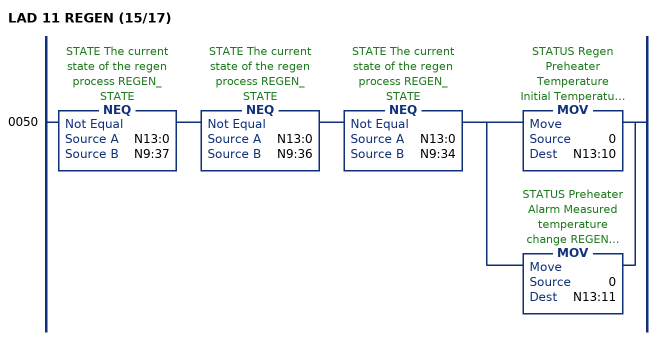
% Rung: 50 %
SOR NEQ N13:0 N9:37 NEQ N13:0 N9:36 NEQ N13:0 N9:34 BST MOV 0 N13:10 NXB MOV 0 N13:11 BND EOR
%   N13:0  REGEN_STATE  "STATE The current state of the regen process" %
%   N9:37  REGEN_ALARM  "STATE Regen Alarm" %
%   N9:36  REGEN_COOL  "STATE Regen Cool" %
%   N9:34  REGEN_RUN  "STATE Regen Running" %
%   N13:10  REGEN_HRS_LEFT  "STATUS Regen Preheater Temperature Initial Temperature" %
%   N13:11  REGEN_MIN_LEFT  "STATUS Preheater Alarm Measured temperature change" %

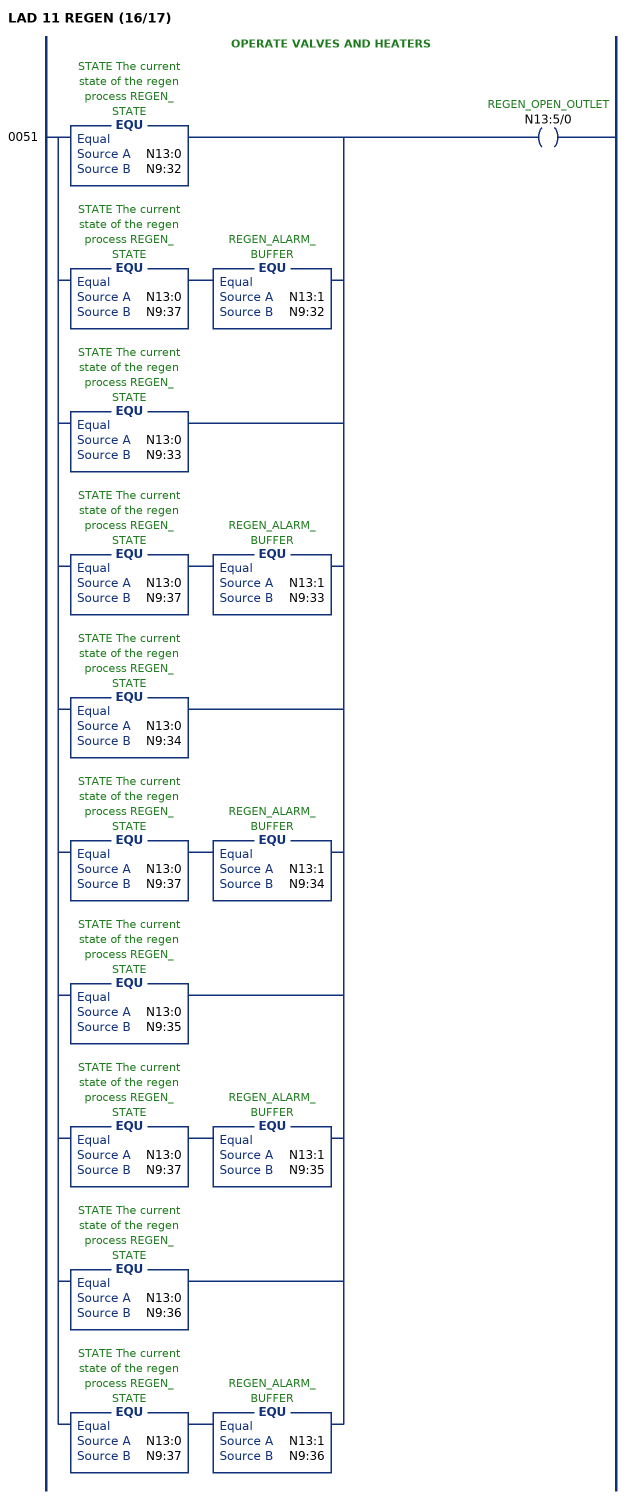
% Rung: 51 %
% TITLE: OPERATE VALVES AND HEATERS %
SOR BST EQU N13:0 N9:32 NXB EQU N13:0 N9:37 EQU N13:1 N9:32 NXB EQU N13:0 N9:33 NXB EQU N13:0 N9:37 EQU N13:1 N9:33 NXB EQU N13:0 N9:34 NXB EQU N13:0 N9:37 EQU N13:1 N9:34 NXB EQU N13:0 N9:35 NXB EQU N13:0 N9:37 EQU N13:1 N9:35 NXB EQU N13:0 N9:36 NXB EQU N13:0 N9:37 EQU N13:1 N9:36 BND OTE N13:5/0 EOR
%   N13:0  REGEN_STATE  "STATE The current state of the regen process" %
%   N9:32  REGEN_VENT  "STATE Regen Vent" %
%   N9:37  REGEN_ALARM  "STATE Regen Alarm" %
%   N13:1  REGEN_ALARM_BUFFER %
%   N9:33  REGEN_HEAT_BED  "STATE Regen Heat wall" %
%   N9:34  REGEN_RUN  "STATE Regen Running" %
%   N9:35  REGEN_COOL_WALL  "STATE Regen Cool wall" %
%   N9:36  REGEN_COOL  "STATE Regen Cool" %
%   N13:5/0  REGEN_OPEN_OUTLET %

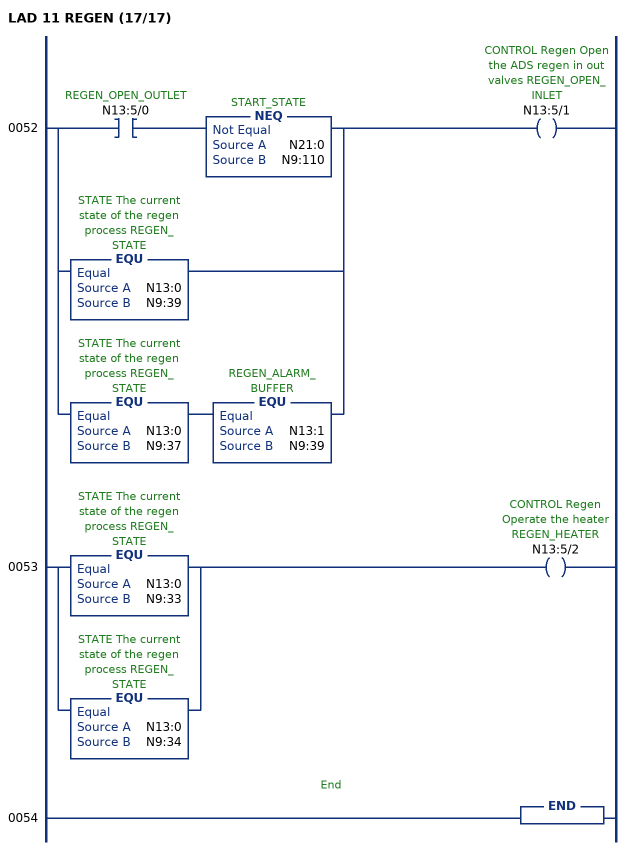
% Rung: 52 %
SOR BST XIC N13:5/0 NEQ N21:0 N9:110 NXB EQU N13:0 N9:39 NXB EQU N13:0 N9:37 EQU N13:1 N9:39 BND OTE N13:5/1 EOR
%   N13:5/0  REGEN_OPEN_OUTLET %
%   N21:0  START_STATE %
%   N9:110  START_REG_VENT %
%   N13:0  REGEN_STATE  "STATE The current state of the regen process" %
%   N9:39  REGEN_BACKFILL %
%   N9:37  REGEN_ALARM  "STATE Regen Alarm" %
%   N13:1  REGEN_ALARM_BUFFER %
%   N13:5/1  REGEN_OPEN_INLET  "CONTROL Regen Open the ADS regen in out valves" %
% Rung: 53 %
SOR BST EQU N13:0 N9:33 NXB EQU N13:0 N9:34 BND OTE N13:5/2 EOR
%   N13:0  REGEN_STATE  "STATE The current state of the regen process" %
%   N9:33  REGEN_HEAT_BED  "STATE Regen Heat wall" %
%   N9:34  REGEN_RUN  "STATE Regen Running" %
%   N13:5/2  REGEN_HEATER  "CONTROL Regen Operate the heater" %
% Rung: 54 %
% End %
SOR END EOR

LADDER 12 "REGEN_FLT"    % regen alarms and warnings %
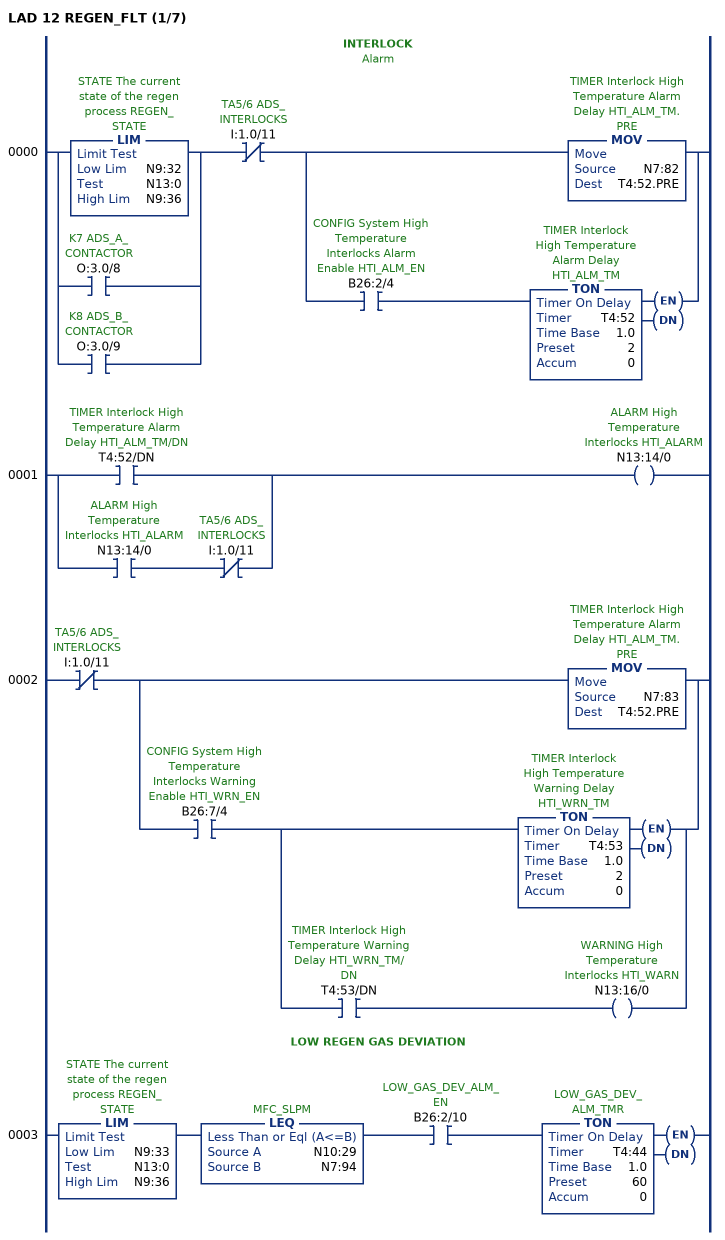
% Rung: 0 %
% TITLE: INTERLOCK %
% Alarm %
SOR BST LIM N9:32 N13:0 N9:36 NXB XIC O:3.0/8 NXB XIC O:3.0/9 BND XIO I:1.0/11 BST MOV N7:82 T4:52.PRE NXB XIC B26:2/4 TON T4:52 1.0 2 0 BND EOR
%   N9:32  REGEN_VENT  "STATE Regen Vent" %
%   N13:0  REGEN_STATE  "STATE The current state of the regen process" %
%   N9:36  REGEN_COOL  "STATE Regen Cool" %
%   O:3.0/8  ADS_A_CONTACTOR  "K7" %
%   O:3.0/9  ADS_B_CONTACTOR  "K8" %
%   I:1.0/11  ADS_INTERLOCKS  "TA5/6" %
%   N7:82  HTI_ALM_DY  "CONFIG Interlocks High Temp Alarm Delay" %
%   T4:52  HTI_ALM_TM  "TIMER Interlock High Temperature Alarm Delay" %
%   B26:2/4  HTI_ALM_EN  "CONFIG System High Temperature Interlocks Alarm Enable" %
% Rung: 1 %
SOR BST XIC T4:52/DN NXB XIC N13:14/0 XIO I:1.0/11 BND OTE N13:14/0 EOR
%   T4:52  HTI_ALM_TM  "TIMER Interlock High Temperature Alarm Delay" %
%   N13:14/0  HTI_ALARM  "ALARM High Temperature Interlocks" %
%   I:1.0/11  ADS_INTERLOCKS  "TA5/6" %
% Rung: 2 %
SOR XIO I:1.0/11 BST MOV N7:83 T4:52.PRE NXB XIC B26:7/4 BST TON T4:53 1.0 2 0 NXB XIC T4:53/DN OTE N13:16/0 BND BND EOR
%   I:1.0/11  ADS_INTERLOCKS  "TA5/6" %
%   N7:83  HTI_WRN_DY  "CONFIG Interlocks High Temp Warning Delay" %
%   T4:52  HTI_ALM_TM  "TIMER Interlock High Temperature Alarm Delay" %
%   B26:7/4  HTI_WRN_EN  "CONFIG System High Temperature Interlocks Warning Enable" %
%   T4:53  HTI_WRN_TM  "TIMER Interlock High Temperature Warning Delay" %
%   N13:16/0  HTI_WARN  "WARNING High Temperature Interlocks" %
% Rung: 3 %
% TITLE: LOW REGEN GAS DEVIATION %
SOR LIM N9:33 N13:0 N9:36 LEQ N10:29 N7:94 XIC B26:2/10 TON T4:44 1.0 60 0 EOR
%   N9:33  REGEN_HEAT_BED  "STATE Regen Heat wall" %
%   N13:0  REGEN_STATE  "STATE The current state of the regen process" %
%   N9:36  REGEN_COOL  "STATE Regen Cool" %
%   N10:29  MFC_SLPM %
%   N7:94  LOW_GAS_DEV_ALM_SP %
%   B26:2/10  LOW_GAS_DEV_ALM_EN %
%   T4:44  LOW_GAS_DEV_ALM_TMR %

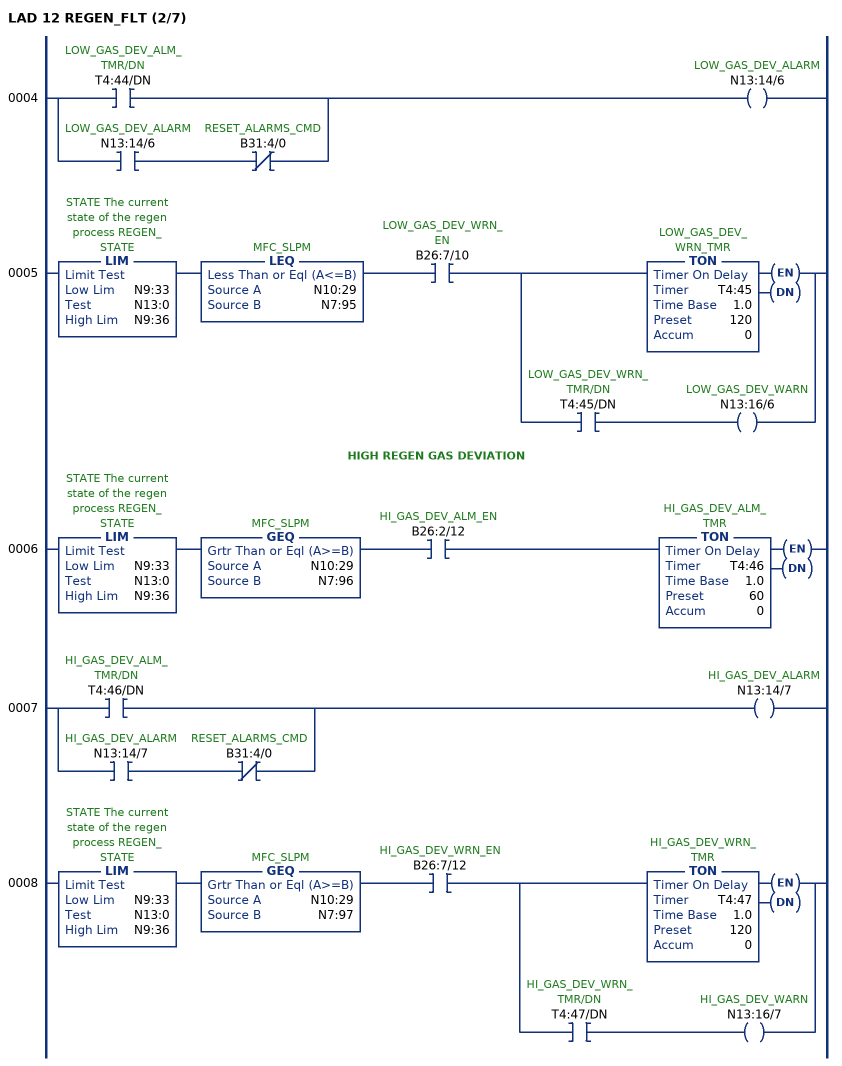
% Rung: 4 %
SOR BST XIC T4:44/DN NXB XIC N13:14/6 XIO B31:4/0 BND OTE N13:14/6 EOR
%   T4:44  LOW_GAS_DEV_ALM_TMR %
%   N13:14/6  LOW_GAS_DEV_ALARM %
%   B31:4/0  RESET_ALARMS_CMD %
% Rung: 5 %
SOR LIM N9:33 N13:0 N9:36 LEQ N10:29 N7:95 XIC B26:7/10 BST TON T4:45 1.0 120 0 NXB XIC T4:45/DN OTE N13:16/6 BND EOR
%   N9:33  REGEN_HEAT_BED  "STATE Regen Heat wall" %
%   N13:0  REGEN_STATE  "STATE The current state of the regen process" %
%   N9:36  REGEN_COOL  "STATE Regen Cool" %
%   N10:29  MFC_SLPM %
%   N7:95  LOW_GAS_DEV_WRN_SP %
%   B26:7/10  LOW_GAS_DEV_WRN_EN %
%   T4:45  LOW_GAS_DEV_WRN_TMR %
%   N13:16/6  LOW_GAS_DEV_WARN %
% Rung: 6 %
% TITLE: HIGH REGEN GAS DEVIATION %
SOR LIM N9:33 N13:0 N9:36 GEQ N10:29 N7:96 XIC B26:2/12 TON T4:46 1.0 60 0 EOR
%   N9:33  REGEN_HEAT_BED  "STATE Regen Heat wall" %
%   N13:0  REGEN_STATE  "STATE The current state of the regen process" %
%   N9:36  REGEN_COOL  "STATE Regen Cool" %
%   N10:29  MFC_SLPM %
%   N7:96  HI_GAS_DEV_ALM_SP %
%   B26:2/12  HI_GAS_DEV_ALM_EN %
%   T4:46  HI_GAS_DEV_ALM_TMR %
% Rung: 7 %
SOR BST XIC T4:46/DN NXB XIC N13:14/7 XIO B31:4/0 BND OTE N13:14/7 EOR
%   T4:46  HI_GAS_DEV_ALM_TMR %
%   N13:14/7  HI_GAS_DEV_ALARM %
%   B31:4/0  RESET_ALARMS_CMD %
% Rung: 8 %
SOR LIM N9:33 N13:0 N9:36 GEQ N10:29 N7:97 XIC B26:7/12 BST TON T4:47 1.0 120 0 NXB XIC T4:47/DN OTE N13:16/7 BND EOR
%   N9:33  REGEN_HEAT_BED  "STATE Regen Heat wall" %
%   N13:0  REGEN_STATE  "STATE The current state of the regen process" %
%   N9:36  REGEN_COOL  "STATE Regen Cool" %
%   N10:29  MFC_SLPM %
%   N7:97  HI_GAS_DEV_WRN_SP %
%   B26:7/12  HI_GAS_DEV_WRN_EN %
%   T4:47  HI_GAS_DEV_WRN_TMR %
%   N13:16/7  HI_GAS_DEV_WARN %

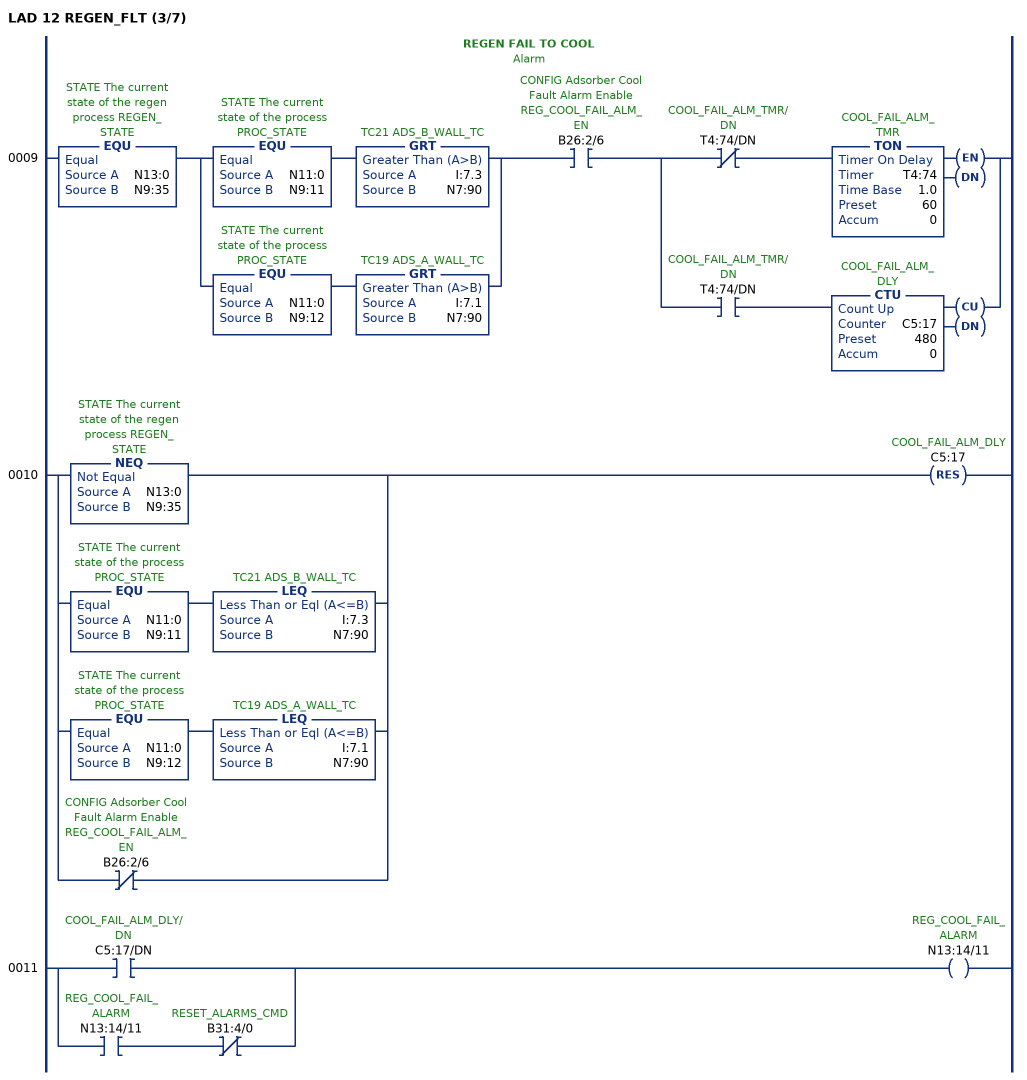
% Rung: 9 %
% TITLE: REGEN FAIL TO COOL %
% Alarm %
SOR EQU N13:0 N9:35 BST EQU N11:0 N9:11 GRT I:7.3 N7:90 NXB EQU N11:0 N9:12 GRT I:7.1 N7:90 BND XIC B26:2/6 BST XIO T4:74/DN TON T4:74 1.0 60 0 NXB XIC T4:74/DN CTU C5:17 480 0 BND EOR
%   N13:0  REGEN_STATE  "STATE The current state of the regen process" %
%   N9:35  REGEN_COOL_WALL  "STATE Regen Cool wall" %
%   N11:0  PROC_STATE  "STATE The current state of the process" %
%   N9:11  PROC_PFY_A_REG_B  "STATE Process Purify A" %
%   I:7.3  ADS_B_WALL_TC  "TC21" %
%   N7:90  REG_COOL_FAIL_ALM_SP %
%   N9:12  PROC_PFY_B_REG_A  "STATE Process Purify B" %
%   I:7.1  ADS_A_WALL_TC  "TC19" %
%   B26:2/6  REG_COOL_FAIL_ALM_EN  "CONFIG Adsorber Cool Fault Alarm Enable" %
%   T4:74  COOL_FAIL_ALM_TMR %
%   C5:17  COOL_FAIL_ALM_DLY %
% Rung: 10 %
SOR BST NEQ N13:0 N9:35 NXB EQU N11:0 N9:11 LEQ I:7.3 N7:90 NXB EQU N11:0 N9:12 LEQ I:7.1 N7:90 NXB XIO B26:2/6 BND RES C5:17 EOR
%   N13:0  REGEN_STATE  "STATE The current state of the regen process" %
%   N9:35  REGEN_COOL_WALL  "STATE Regen Cool wall" %
%   N11:0  PROC_STATE  "STATE The current state of the process" %
%   N9:11  PROC_PFY_A_REG_B  "STATE Process Purify A" %
%   I:7.3  ADS_B_WALL_TC  "TC21" %
%   N7:90  REG_COOL_FAIL_ALM_SP %
%   N9:12  PROC_PFY_B_REG_A  "STATE Process Purify B" %
%   I:7.1  ADS_A_WALL_TC  "TC19" %
%   B26:2/6  REG_COOL_FAIL_ALM_EN  "CONFIG Adsorber Cool Fault Alarm Enable" %
%   C5:17  COOL_FAIL_ALM_DLY %
% Rung: 11 %
SOR BST XIC C5:17/DN NXB XIC N13:14/11 XIO B31:4/0 BND OTE N13:14/11 EOR
%   C5:17  COOL_FAIL_ALM_DLY %
%   N13:14/11  REG_COOL_FAIL_ALARM %
%   B31:4/0  RESET_ALARMS_CMD %

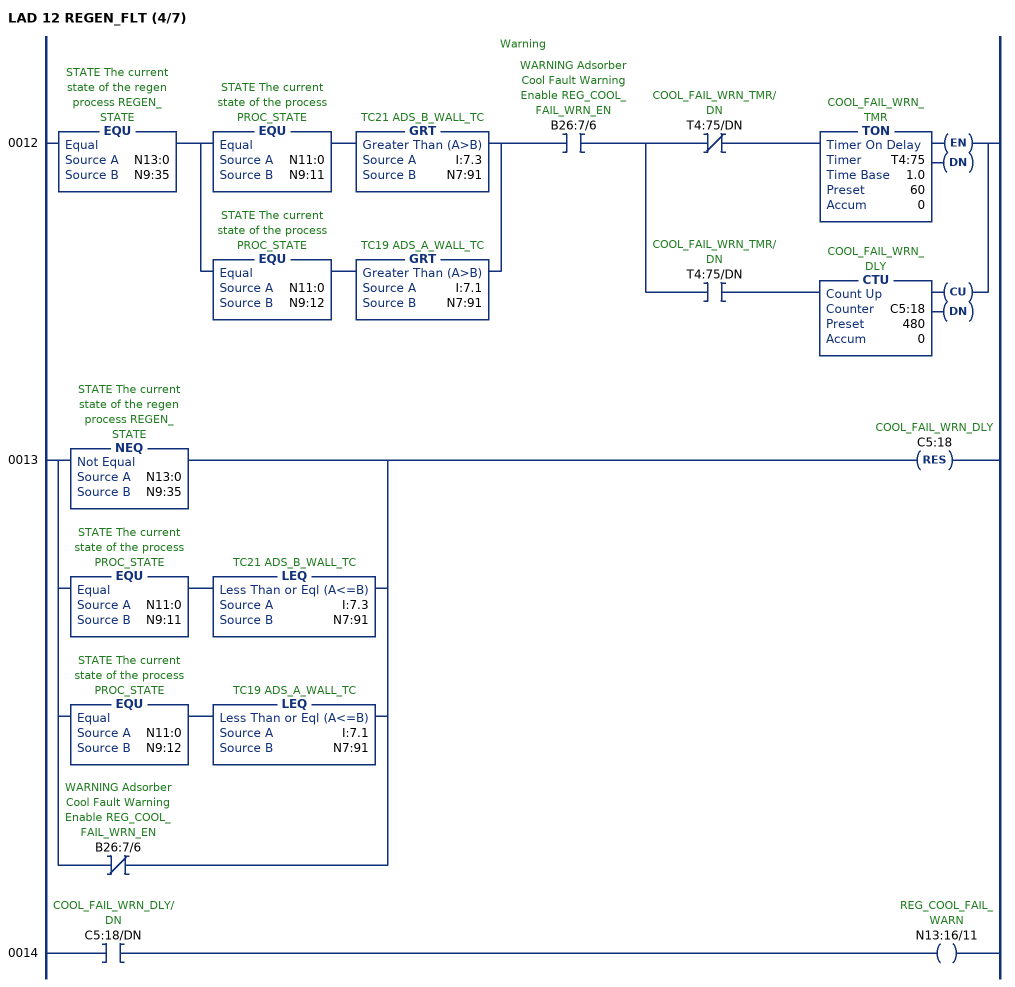
% Rung: 12 %
% Warning %
SOR EQU N13:0 N9:35 BST EQU N11:0 N9:11 GRT I:7.3 N7:91 NXB EQU N11:0 N9:12 GRT I:7.1 N7:91 BND XIC B26:7/6 BST XIO T4:75/DN TON T4:75 1.0 60 0 NXB XIC T4:75/DN CTU C5:18 480 0 BND EOR
%   N13:0  REGEN_STATE  "STATE The current state of the regen process" %
%   N9:35  REGEN_COOL_WALL  "STATE Regen Cool wall" %
%   N11:0  PROC_STATE  "STATE The current state of the process" %
%   N9:11  PROC_PFY_A_REG_B  "STATE Process Purify A" %
%   I:7.3  ADS_B_WALL_TC  "TC21" %
%   N7:91  REG_COOL_FAIL_WRN_SP %
%   N9:12  PROC_PFY_B_REG_A  "STATE Process Purify B" %
%   I:7.1  ADS_A_WALL_TC  "TC19" %
%   B26:7/6  REG_COOL_FAIL_WRN_EN  "WARNING Adsorber Cool Fault Warning Enable" %
%   T4:75  COOL_FAIL_WRN_TMR %
%   C5:18  COOL_FAIL_WRN_DLY %
% Rung: 13 %
SOR BST NEQ N13:0 N9:35 NXB EQU N11:0 N9:11 LEQ I:7.3 N7:91 NXB EQU N11:0 N9:12 LEQ I:7.1 N7:91 NXB XIO B26:7/6 BND RES C5:18 EOR
%   N13:0  REGEN_STATE  "STATE The current state of the regen process" %
%   N9:35  REGEN_COOL_WALL  "STATE Regen Cool wall" %
%   N11:0  PROC_STATE  "STATE The current state of the process" %
%   N9:11  PROC_PFY_A_REG_B  "STATE Process Purify A" %
%   I:7.3  ADS_B_WALL_TC  "TC21" %
%   N7:91  REG_COOL_FAIL_WRN_SP %
%   N9:12  PROC_PFY_B_REG_A  "STATE Process Purify B" %
%   I:7.1  ADS_A_WALL_TC  "TC19" %
%   B26:7/6  REG_COOL_FAIL_WRN_EN  "WARNING Adsorber Cool Fault Warning Enable" %
%   C5:18  COOL_FAIL_WRN_DLY %
% Rung: 14 %
SOR XIC C5:18/DN OTE N13:16/11 EOR
%   C5:18  COOL_FAIL_WRN_DLY %
%   N13:16/11  REG_COOL_FAIL_WARN %

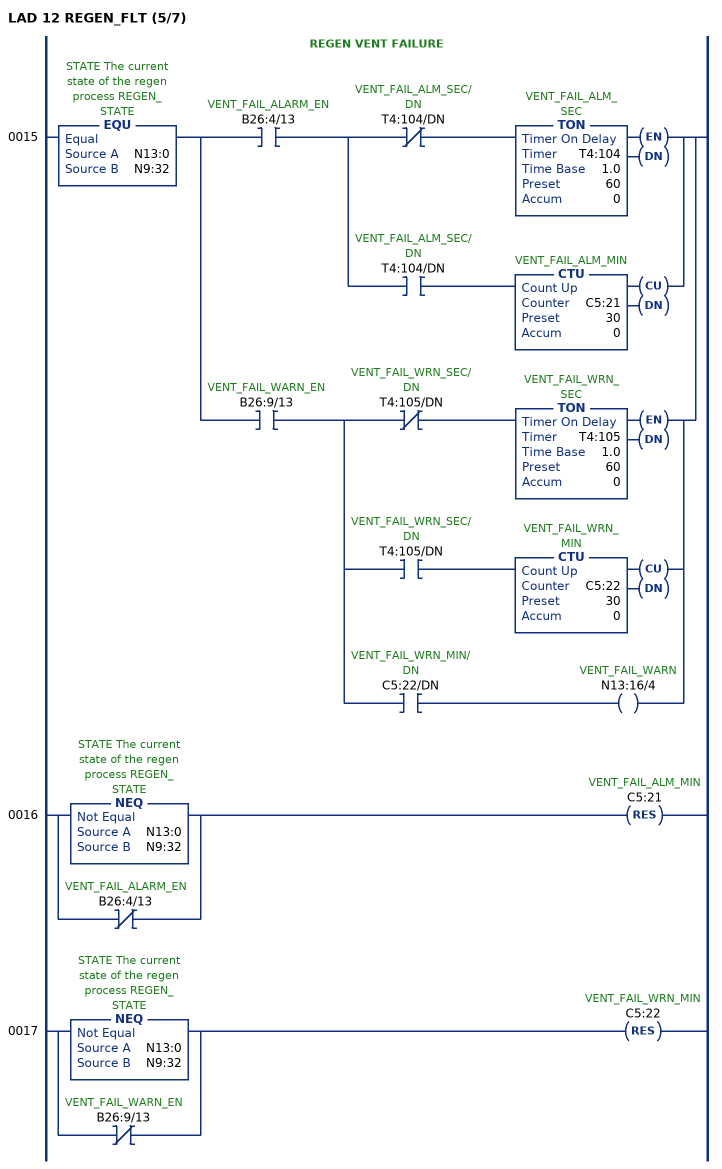
% Rung: 15 %
% TITLE: REGEN VENT FAILURE %
SOR EQU N13:0 N9:32 BST XIC B26:4/13 BST XIO T4:104/DN TON T4:104 1.0 60 0 NXB XIC T4:104/DN CTU C5:21 30 0 BND NXB XIC B26:9/13 BST XIO T4:105/DN TON T4:105 1.0 60 0 NXB XIC T4:105/DN CTU C5:22 30 0 NXB XIC C5:22/DN OTE N13:16/4 BND BND EOR
%   N13:0  REGEN_STATE  "STATE The current state of the regen process" %
%   N9:32  REGEN_VENT  "STATE Regen Vent" %
%   B26:4/13  VENT_FAIL_ALARM_EN %
%   T4:104  VENT_FAIL_ALM_SEC %
%   C5:21  VENT_FAIL_ALM_MIN %
%   B26:9/13  VENT_FAIL_WARN_EN %
%   T4:105  VENT_FAIL_WRN_SEC %
%   C5:22  VENT_FAIL_WRN_MIN %
%   N13:16/4  VENT_FAIL_WARN %
% Rung: 16 %
SOR BST NEQ N13:0 N9:32 NXB XIO B26:4/13 BND RES C5:21 EOR
%   N13:0  REGEN_STATE  "STATE The current state of the regen process" %
%   N9:32  REGEN_VENT  "STATE Regen Vent" %
%   B26:4/13  VENT_FAIL_ALARM_EN %
%   C5:21  VENT_FAIL_ALM_MIN %
% Rung: 17 %
SOR BST NEQ N13:0 N9:32 NXB XIO B26:9/13 BND RES C5:22 EOR
%   N13:0  REGEN_STATE  "STATE The current state of the regen process" %
%   N9:32  REGEN_VENT  "STATE Regen Vent" %
%   B26:9/13  VENT_FAIL_WARN_EN %
%   C5:22  VENT_FAIL_WRN_MIN %

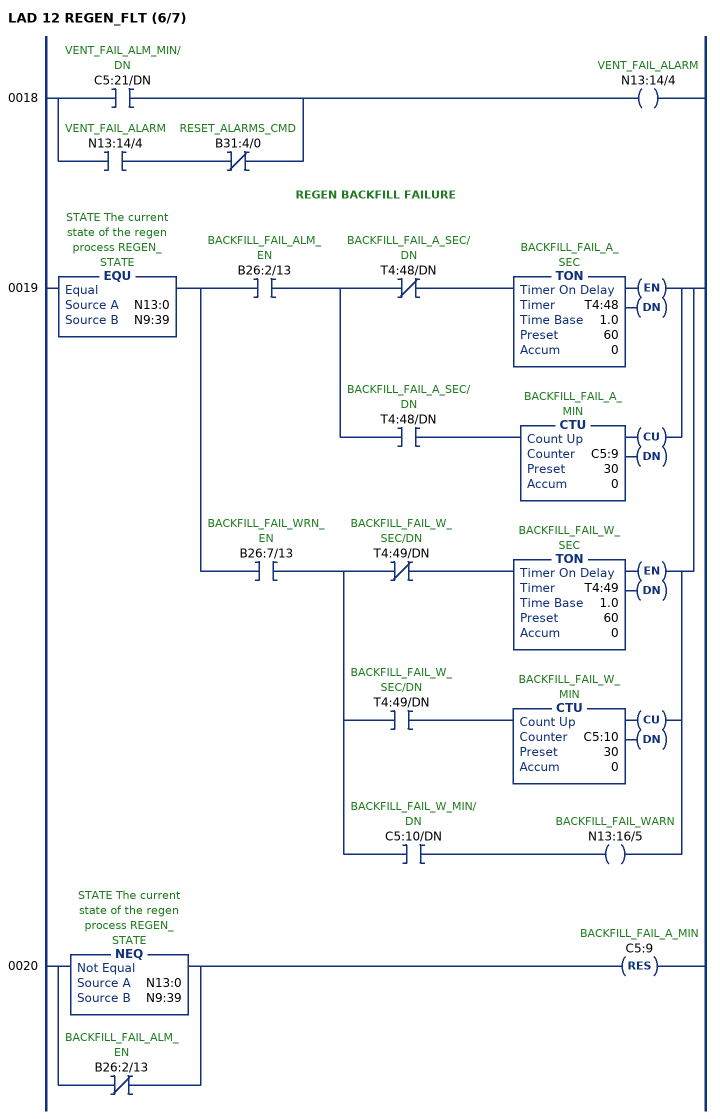
% Rung: 18 %
SOR BST XIC C5:21/DN NXB XIC N13:14/4 XIO B31:4/0 BND OTE N13:14/4 EOR
%   C5:21  VENT_FAIL_ALM_MIN %
%   N13:14/4  VENT_FAIL_ALARM %
%   B31:4/0  RESET_ALARMS_CMD %
% Rung: 19 %
% TITLE: REGEN BACKFILL FAILURE %
SOR EQU N13:0 N9:39 BST XIC B26:2/13 BST XIO T4:48/DN TON T4:48 1.0 60 0 NXB XIC T4:48/DN CTU C5:9 30 0 BND NXB XIC B26:7/13 BST XIO T4:49/DN TON T4:49 1.0 60 0 NXB XIC T4:49/DN CTU C5:10 30 0 NXB XIC C5:10/DN OTE N13:16/5 BND BND EOR
%   N13:0  REGEN_STATE  "STATE The current state of the regen process" %
%   N9:39  REGEN_BACKFILL %
%   B26:2/13  BACKFILL_FAIL_ALM_EN %
%   T4:48  BACKFILL_FAIL_A_SEC %
%   C5:9  BACKFILL_FAIL_A_MIN %
%   B26:7/13  BACKFILL_FAIL_WRN_EN %
%   T4:49  BACKFILL_FAIL_W_SEC %
%   C5:10  BACKFILL_FAIL_W_MIN %
%   N13:16/5  BACKFILL_FAIL_WARN %
% Rung: 20 %
SOR BST NEQ N13:0 N9:39 NXB XIO B26:2/13 BND RES C5:9 EOR
%   N13:0  REGEN_STATE  "STATE The current state of the regen process" %
%   N9:39  REGEN_BACKFILL %
%   B26:2/13  BACKFILL_FAIL_ALM_EN %
%   C5:9  BACKFILL_FAIL_A_MIN %

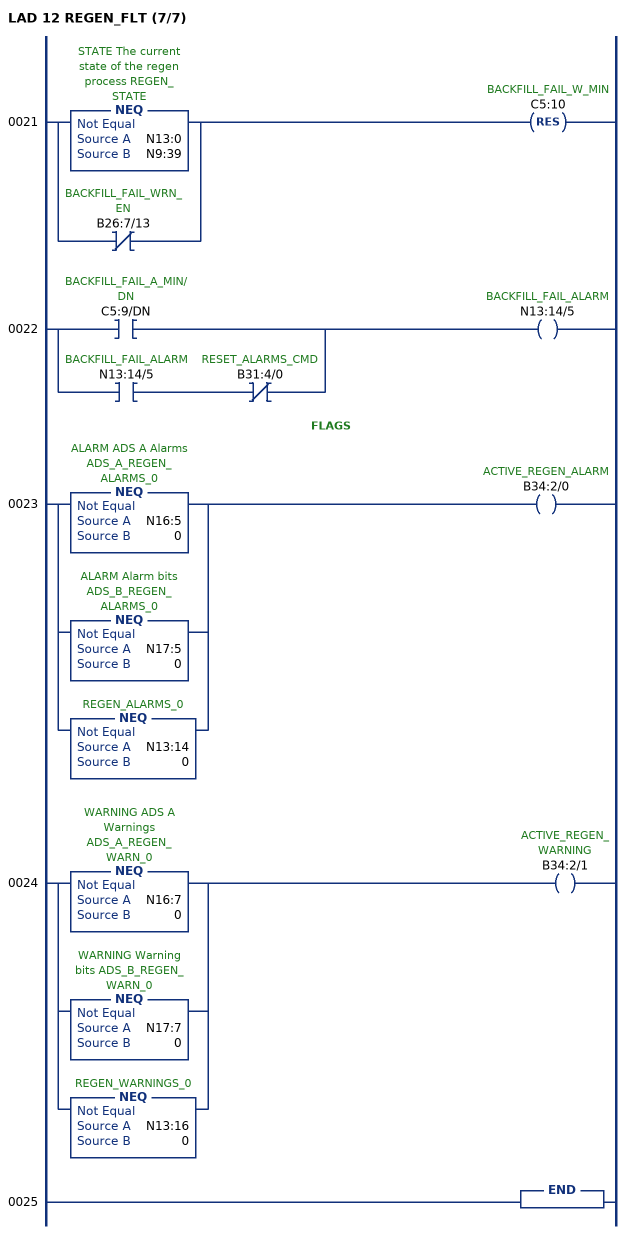
% Rung: 21 %
SOR BST NEQ N13:0 N9:39 NXB XIO B26:7/13 BND RES C5:10 EOR
%   N13:0  REGEN_STATE  "STATE The current state of the regen process" %
%   N9:39  REGEN_BACKFILL %
%   B26:7/13  BACKFILL_FAIL_WRN_EN %
%   C5:10  BACKFILL_FAIL_W_MIN %
% Rung: 22 %
SOR BST XIC C5:9/DN NXB XIC N13:14/5 XIO B31:4/0 BND OTE N13:14/5 EOR
%   C5:9  BACKFILL_FAIL_A_MIN %
%   N13:14/5  BACKFILL_FAIL_ALARM %
%   B31:4/0  RESET_ALARMS_CMD %
% Rung: 23 %
% TITLE: FLAGS %
SOR BST NEQ N16:5 0 NXB NEQ N17:5 0 NXB NEQ N13:14 0 BND OTE B34:2/0 EOR
%   N16:5  ADS_A_REGEN_ALARMS_0  "ALARM ADS A Alarms" %
%   N17:5  ADS_B_REGEN_ALARMS_0  "ALARM Alarm bits" %
%   N13:14  REGEN_ALARMS_0 %
%   B34:2/0  ACTIVE_REGEN_ALARM %
% Rung: 24 %
SOR BST NEQ N16:7 0 NXB NEQ N17:7 0 NXB NEQ N13:16 0 BND OTE B34:2/1 EOR
%   N16:7  ADS_A_REGEN_WARN_0  "WARNING ADS A Warnings" %
%   N17:7  ADS_B_REGEN_WARN_0  "WARNING Warning bits" %
%   N13:16  REGEN_WARNINGS_0 %
%   B34:2/1  ACTIVE_REGEN_WARNING %
% Rung: 25 %
SOR END EOR

LADDER 13 "PURGE"
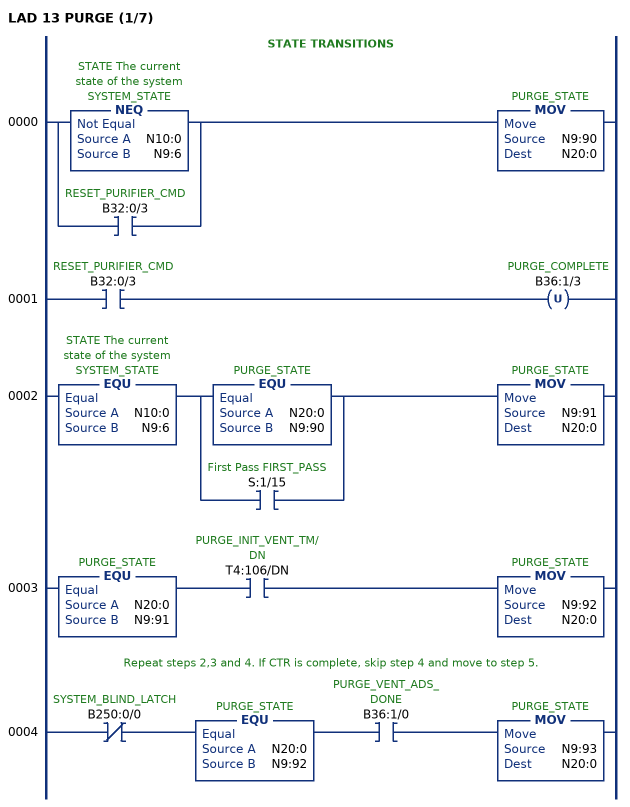
% Rung: 0 %
% TITLE: STATE TRANSITIONS %
SOR BST NEQ N10:0 N9:6 NXB XIC B32:0/3 BND MOV N9:90 N20:0 EOR
%   N10:0  SYSTEM_STATE  "STATE The current state of the system" %
%   N9:6  SYSTEM_PURGE %
%   B32:0/3  RESET_PURIFIER_CMD %
%   N9:90  PURGE_IDLE %
%   N20:0  PURGE_STATE %
% Rung: 1 %
SOR XIC B32:0/3 OTU B36:1/3 EOR
%   B32:0/3  RESET_PURIFIER_CMD %
%   B36:1/3  PURGE_COMPLETE %
% Rung: 2 %
SOR EQU N10:0 N9:6 BST EQU N20:0 N9:90 NXB XIC S:1/15 BND MOV N9:91 N20:0 EOR
%   N10:0  SYSTEM_STATE  "STATE The current state of the system" %
%   N9:6  SYSTEM_PURGE %
%   N20:0  PURGE_STATE %
%   N9:90  PURGE_IDLE %
%   S:1/15  FIRST_PASS  "First Pass" %
%   N9:91  PURGE_INIT_VENT %
% Rung: 3 %
SOR EQU N20:0 N9:91 XIC T4:106/DN MOV N9:92 N20:0 EOR
%   N20:0  PURGE_STATE %
%   N9:91  PURGE_INIT_VENT %
%   T4:106  PURGE_INIT_VENT_TM %
%   N9:92  PURGE_VENT_ADSORBER %
% Rung: 4 %
% Repeat steps 2,3 and 4. If CTR is complete, skip step 4 and move to step 5. %
SOR XIO B250:0/0 EQU N20:0 N9:92 XIC B36:1/0 MOV N9:93 N20:0 EOR
%   B250:0/0  SYSTEM_BLIND_LATCH %
%   N20:0  PURGE_STATE %
%   N9:92  PURGE_VENT_ADSORBER %
%   B36:1/0  PURGE_VENT_ADS_DONE %
%   N9:93  PURGE_VENT_GETTER %

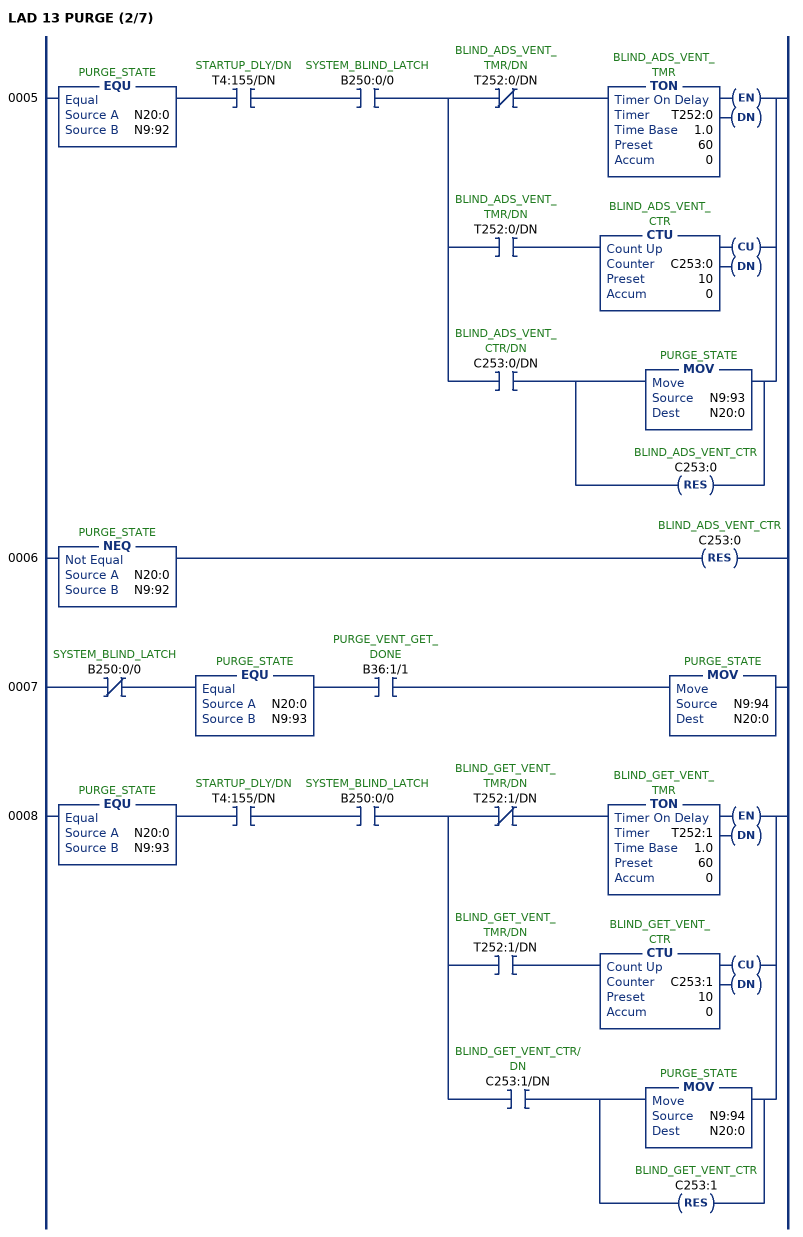
% Rung: 5 %
SOR EQU N20:0 N9:92 XIC T4:155/DN XIC B250:0/0 BST XIO T252:0/DN TON T252:0 1.0 60 0 NXB XIC T252:0/DN CTU C253:0 10 0 NXB XIC C253:0/DN BST MOV N9:93 N20:0 NXB RES C253:0 BND BND EOR
%   N20:0  PURGE_STATE %
%   N9:92  PURGE_VENT_ADSORBER %
%   T4:155  STARTUP_DLY %
%   B250:0/0  SYSTEM_BLIND_LATCH %
%   T252:0  BLIND_ADS_VENT_TMR %
%   C253:0  BLIND_ADS_VENT_CTR %
%   N9:93  PURGE_VENT_GETTER %
% Rung: 6 %
SOR NEQ N20:0 N9:92 RES C253:0 EOR
%   N20:0  PURGE_STATE %
%   N9:92  PURGE_VENT_ADSORBER %
%   C253:0  BLIND_ADS_VENT_CTR %
% Rung: 7 %
SOR XIO B250:0/0 EQU N20:0 N9:93 XIC B36:1/1 MOV N9:94 N20:0 EOR
%   B250:0/0  SYSTEM_BLIND_LATCH %
%   N20:0  PURGE_STATE %
%   N9:93  PURGE_VENT_GETTER %
%   B36:1/1  PURGE_VENT_GET_DONE %
%   N9:94  PURGE_BACKFILL %
% Rung: 8 %
SOR EQU N20:0 N9:93 XIC T4:155/DN XIC B250:0/0 BST XIO T252:1/DN TON T252:1 1.0 60 0 NXB XIC T252:1/DN CTU C253:1 10 0 NXB XIC C253:1/DN BST MOV N9:94 N20:0 NXB RES C253:1 BND BND EOR
%   N20:0  PURGE_STATE %
%   N9:93  PURGE_VENT_GETTER %
%   T4:155  STARTUP_DLY %
%   B250:0/0  SYSTEM_BLIND_LATCH %
%   T252:1  BLIND_GET_VENT_TMR %
%   C253:1  BLIND_GET_VENT_CTR %
%   N9:94  PURGE_BACKFILL %

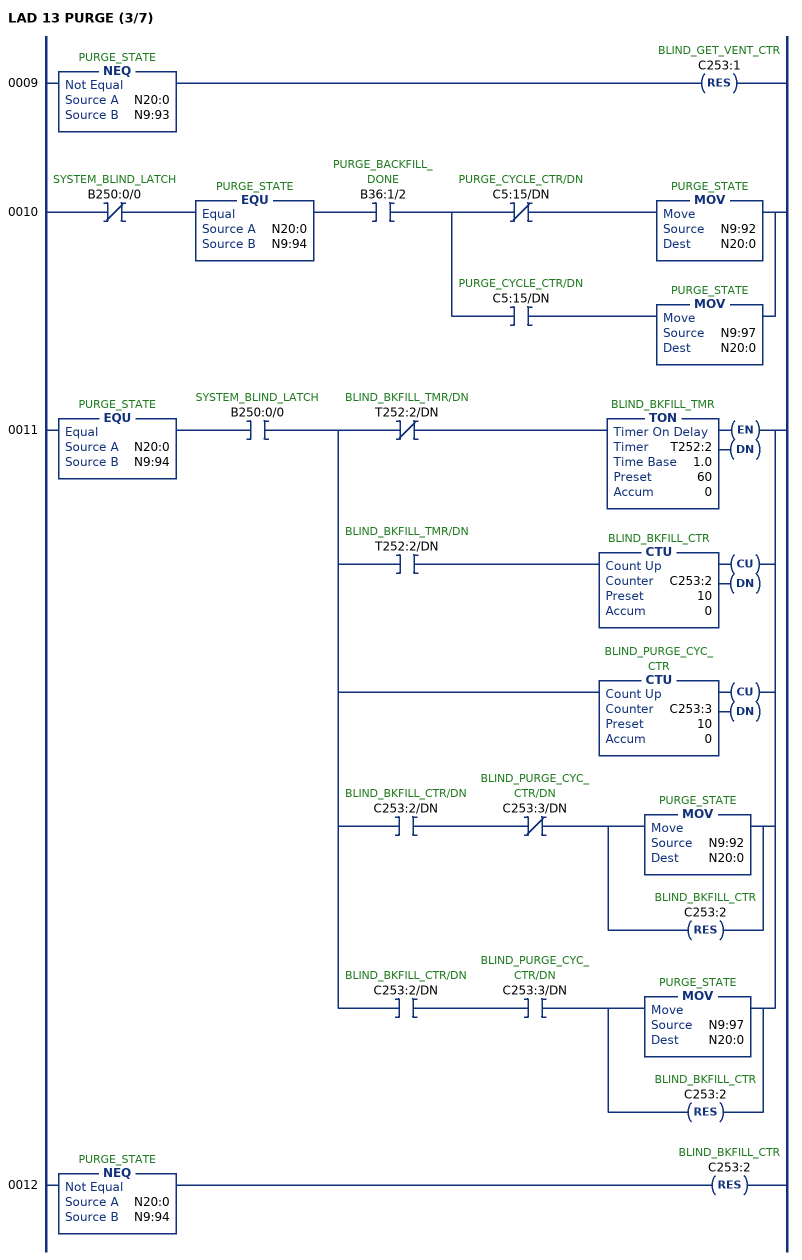
% Rung: 9 %
SOR NEQ N20:0 N9:93 RES C253:1 EOR
%   N20:0  PURGE_STATE %
%   N9:93  PURGE_VENT_GETTER %
%   C253:1  BLIND_GET_VENT_CTR %
% Rung: 10 %
SOR XIO B250:0/0 EQU N20:0 N9:94 XIC B36:1/2 BST XIO C5:15/DN MOV N9:92 N20:0 NXB XIC C5:15/DN MOV N9:97 N20:0 BND EOR
%   B250:0/0  SYSTEM_BLIND_LATCH %
%   N20:0  PURGE_STATE %
%   N9:94  PURGE_BACKFILL %
%   B36:1/2  PURGE_BACKFILL_DONE %
%   C5:15  PURGE_CYCLE_CTR %
%   N9:92  PURGE_VENT_ADSORBER %
%   N9:97  PURGE_VENT_ADS_2 %
% Rung: 11 %
SOR EQU N20:0 N9:94 XIC B250:0/0 BST XIO T252:2/DN TON T252:2 1.0 60 0 NXB XIC T252:2/DN CTU C253:2 10 0 NXB CTU C253:3 10 0 NXB XIC C253:2/DN XIO C253:3/DN BST MOV N9:92 N20:0 NXB RES C253:2 BND NXB XIC C253:2/DN XIC C253:3/DN BST MOV N9:97 N20:0 NXB RES C253:2 BND BND EOR
%   N20:0  PURGE_STATE %
%   N9:94  PURGE_BACKFILL %
%   B250:0/0  SYSTEM_BLIND_LATCH %
%   T252:2  BLIND_BKFILL_TMR %
%   C253:2  BLIND_BKFILL_CTR %
%   C253:3  BLIND_PURGE_CYC_CTR %
%   N9:92  PURGE_VENT_ADSORBER %
%   N9:97  PURGE_VENT_ADS_2 %
% Rung: 12 %
SOR NEQ N20:0 N9:94 RES C253:2 EOR
%   N20:0  PURGE_STATE %
%   N9:94  PURGE_BACKFILL %
%   C253:2  BLIND_BKFILL_CTR %

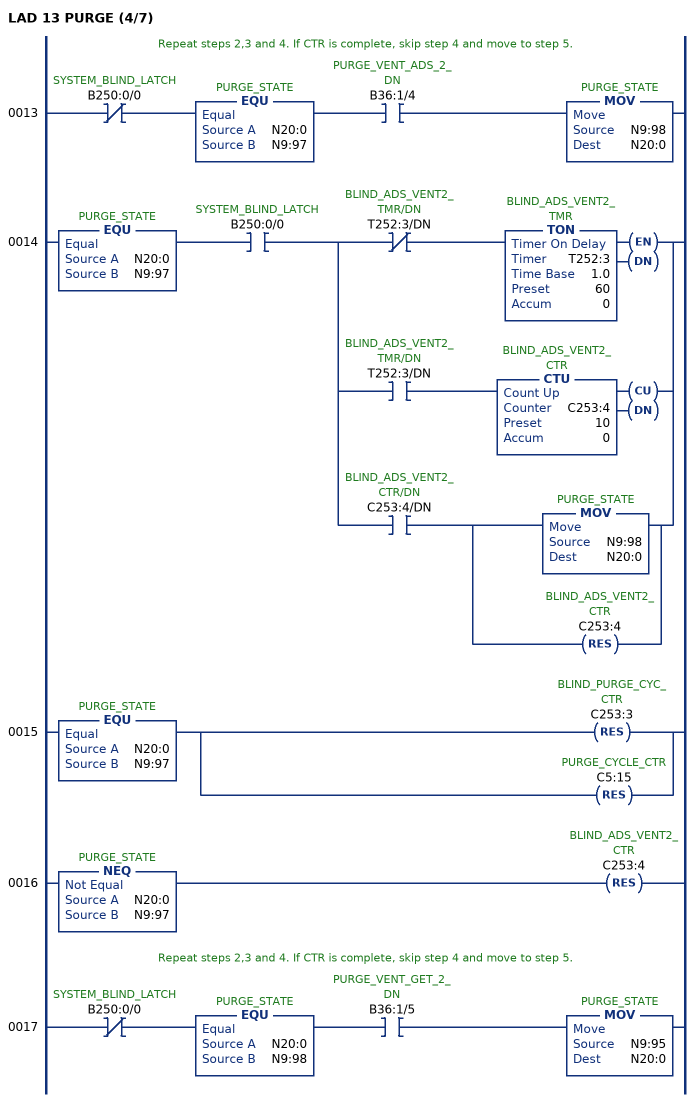
% Rung: 13 %
% Repeat steps 2,3 and 4. If CTR is complete, skip step 4 and move to step 5. %
SOR XIO B250:0/0 EQU N20:0 N9:97 XIC B36:1/4 MOV N9:98 N20:0 EOR
%   B250:0/0  SYSTEM_BLIND_LATCH %
%   N20:0  PURGE_STATE %
%   N9:97  PURGE_VENT_ADS_2 %
%   B36:1/4  PURGE_VENT_ADS_2_DN %
%   N9:98  PURGE_VENT_GET_2 %
% Rung: 14 %
SOR EQU N20:0 N9:97 XIC B250:0/0 BST XIO T252:3/DN TON T252:3 1.0 60 0 NXB XIC T252:3/DN CTU C253:4 10 0 NXB XIC C253:4/DN BST MOV N9:98 N20:0 NXB RES C253:4 BND BND EOR
%   N20:0  PURGE_STATE %
%   N9:97  PURGE_VENT_ADS_2 %
%   B250:0/0  SYSTEM_BLIND_LATCH %
%   T252:3  BLIND_ADS_VENT2_TMR %
%   C253:4  BLIND_ADS_VENT2_CTR %
%   N9:98  PURGE_VENT_GET_2 %
% Rung: 15 %
SOR EQU N20:0 N9:97 BST RES C253:3 NXB RES C5:15 BND EOR
%   N20:0  PURGE_STATE %
%   N9:97  PURGE_VENT_ADS_2 %
%   C253:3  BLIND_PURGE_CYC_CTR %
%   C5:15  PURGE_CYCLE_CTR %
% Rung: 16 %
SOR NEQ N20:0 N9:97 RES C253:4 EOR
%   N20:0  PURGE_STATE %
%   N9:97  PURGE_VENT_ADS_2 %
%   C253:4  BLIND_ADS_VENT2_CTR %
% Rung: 17 %
% Repeat steps 2,3 and 4. If CTR is complete, skip step 4 and move to step 5. %
SOR XIO B250:0/0 EQU N20:0 N9:98 XIC B36:1/5 MOV N9:95 N20:0 EOR
%   B250:0/0  SYSTEM_BLIND_LATCH %
%   N20:0  PURGE_STATE %
%   N9:98  PURGE_VENT_GET_2 %
%   B36:1/5  PURGE_VENT_GET_2_DN %
%   N9:95  PURGE_FINAL_VENT %

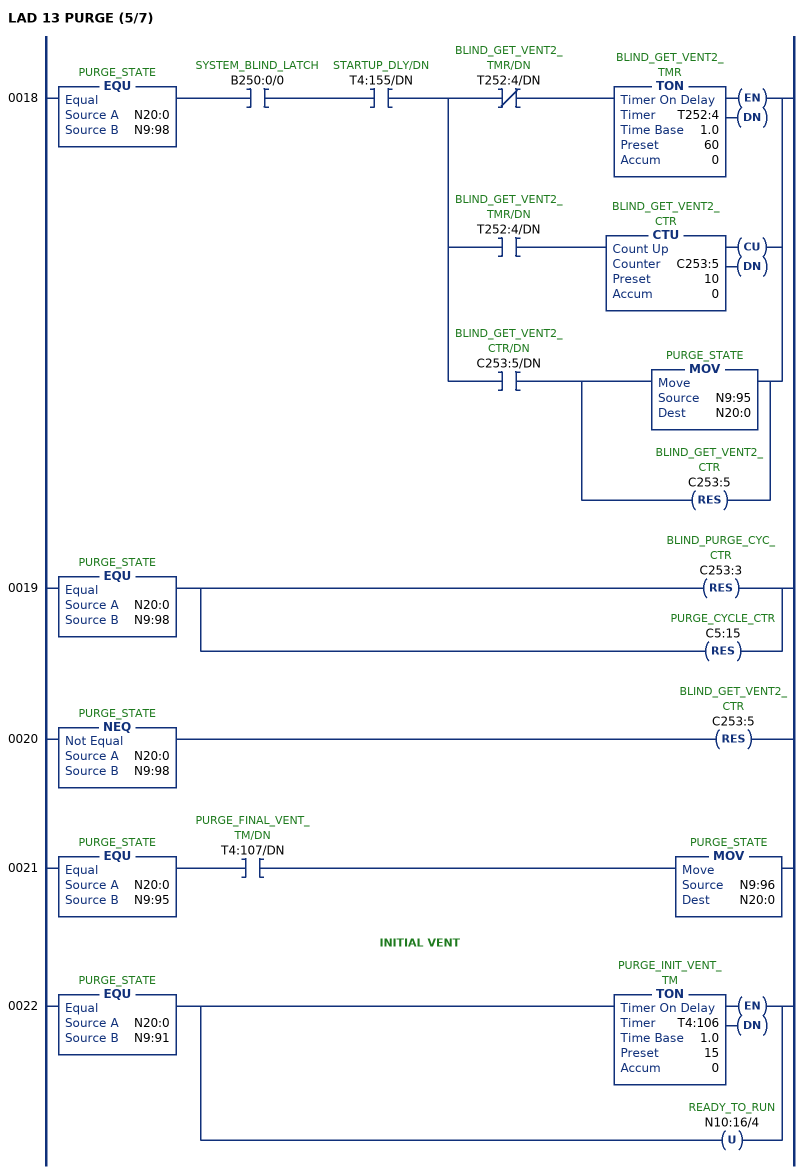
% Rung: 18 %
SOR EQU N20:0 N9:98 XIC B250:0/0 XIC T4:155/DN BST XIO T252:4/DN TON T252:4 1.0 60 0 NXB XIC T252:4/DN CTU C253:5 10 0 NXB XIC C253:5/DN BST MOV N9:95 N20:0 NXB RES C253:5 BND BND EOR
%   N20:0  PURGE_STATE %
%   N9:98  PURGE_VENT_GET_2 %
%   B250:0/0  SYSTEM_BLIND_LATCH %
%   T4:155  STARTUP_DLY %
%   T252:4  BLIND_GET_VENT2_TMR %
%   C253:5  BLIND_GET_VENT2_CTR %
%   N9:95  PURGE_FINAL_VENT %
% Rung: 19 %
SOR EQU N20:0 N9:98 BST RES C253:3 NXB RES C5:15 BND EOR
%   N20:0  PURGE_STATE %
%   N9:98  PURGE_VENT_GET_2 %
%   C253:3  BLIND_PURGE_CYC_CTR %
%   C5:15  PURGE_CYCLE_CTR %
% Rung: 20 %
SOR NEQ N20:0 N9:98 RES C253:5 EOR
%   N20:0  PURGE_STATE %
%   N9:98  PURGE_VENT_GET_2 %
%   C253:5  BLIND_GET_VENT2_CTR %
% Rung: 21 %
SOR EQU N20:0 N9:95 XIC T4:107/DN MOV N9:96 N20:0 EOR
%   N20:0  PURGE_STATE %
%   N9:95  PURGE_FINAL_VENT %
%   T4:107  PURGE_FINAL_VENT_TM %
%   N9:96  PURGE_DONE %
% Rung: 22 %
% TITLE: INITIAL VENT %
SOR EQU N20:0 N9:91 BST TON T4:106 1.0 15 0 NXB OTU N10:16/4 BND EOR
%   N20:0  PURGE_STATE %
%   N9:91  PURGE_INIT_VENT %
%   T4:106  PURGE_INIT_VENT_TM %
%   N10:16/4  READY_TO_RUN %

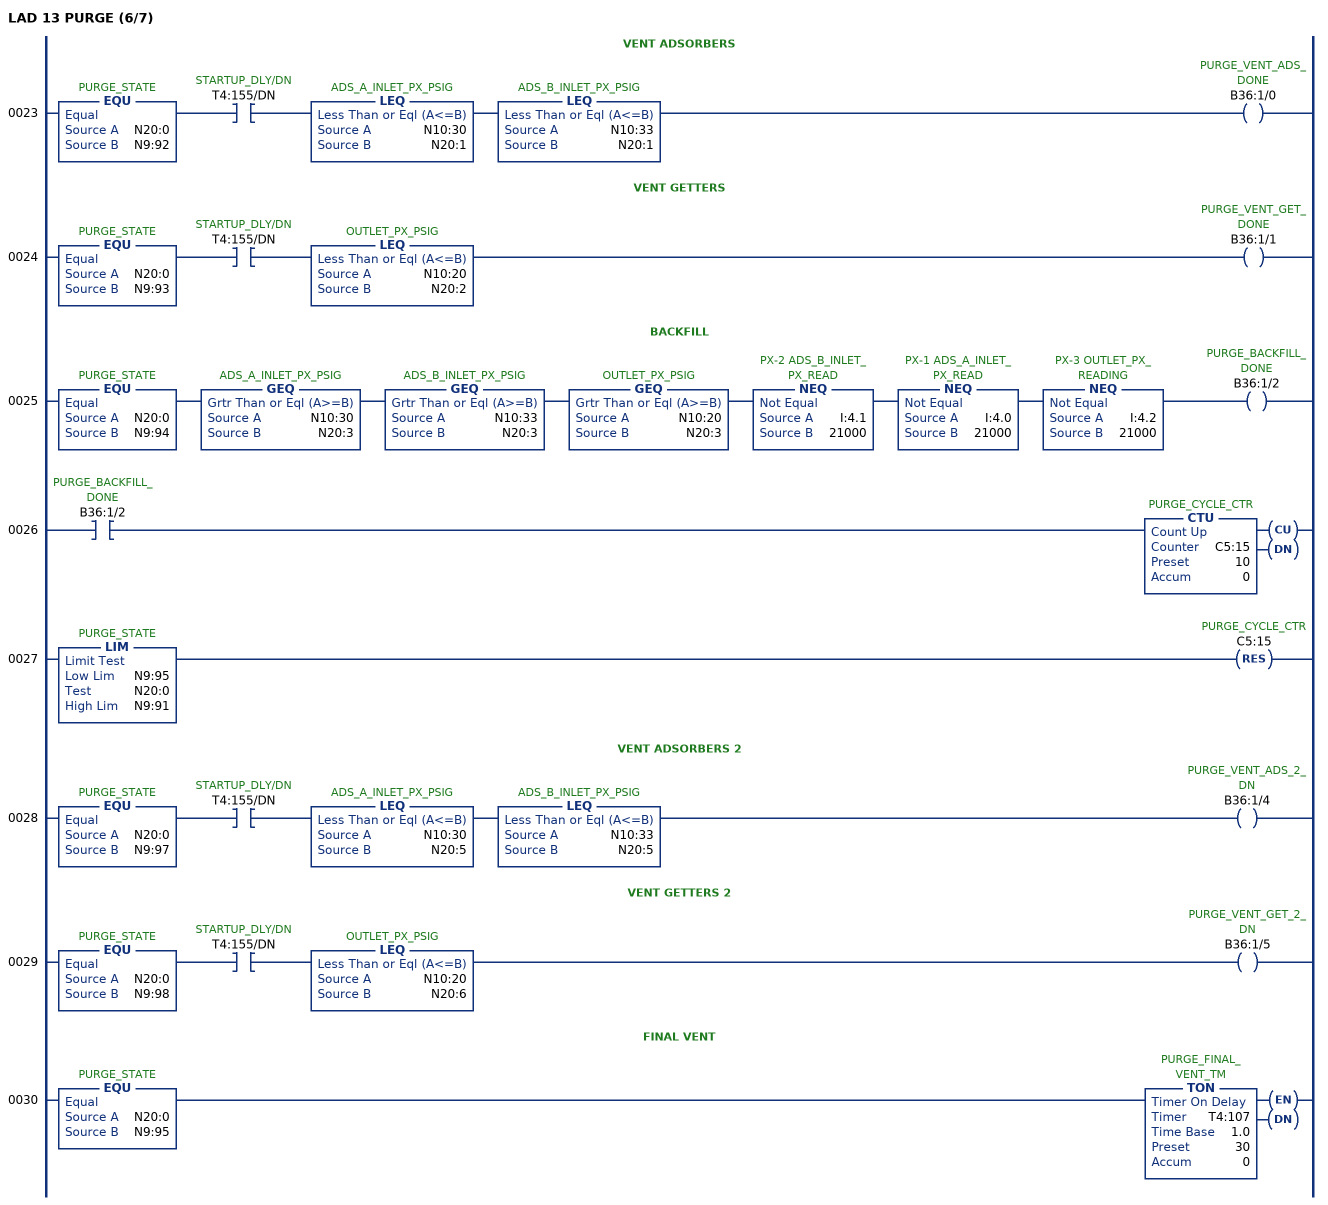
% Rung: 23 %
% TITLE: VENT ADSORBERS %
SOR EQU N20:0 N9:92 XIC T4:155/DN LEQ N10:30 N20:1 LEQ N10:33 N20:1 OTE B36:1/0 EOR
%   N20:0  PURGE_STATE %
%   N9:92  PURGE_VENT_ADSORBER %
%   T4:155  STARTUP_DLY %
%   N10:30  ADS_A_INLET_PX_PSIG %
%   N20:1  PURGE_VENT_ADS_PRES %
%   N10:33  ADS_B_INLET_PX_PSIG %
%   B36:1/0  PURGE_VENT_ADS_DONE %
% Rung: 24 %
% TITLE: VENT GETTERS %
SOR EQU N20:0 N9:93 XIC T4:155/DN LEQ N10:20 N20:2 OTE B36:1/1 EOR
%   N20:0  PURGE_STATE %
%   N9:93  PURGE_VENT_GETTER %
%   T4:155  STARTUP_DLY %
%   N10:20  OUTLET_PX_PSIG %
%   N20:2  PURGE_VENT_GET_PRES %
%   B36:1/1  PURGE_VENT_GET_DONE %
% Rung: 25 %
% TITLE: BACKFILL %
SOR EQU N20:0 N9:94 GEQ N10:30 N20:3 GEQ N10:33 N20:3 GEQ N10:20 N20:3 NEQ I:4.1 21000 NEQ I:4.0 21000 NEQ I:4.2 21000 OTE B36:1/2 EOR
%   N20:0  PURGE_STATE %
%   N9:94  PURGE_BACKFILL %
%   N10:30  ADS_A_INLET_PX_PSIG %
%   N20:3  PURGE_BKFIL_PRES %
%   N10:33  ADS_B_INLET_PX_PSIG %
%   N10:20  OUTLET_PX_PSIG %
%   I:4.1  ADS_B_INLET_PX_READ  "PX-2" %
%   I:4.0  ADS_A_INLET_PX_READ  "PX-1" %
%   I:4.2  OUTLET_PX_READING  "PX-3" %
%   B36:1/2  PURGE_BACKFILL_DONE %
% Rung: 26 %
SOR XIC B36:1/2 CTU C5:15 10 0 EOR
%   B36:1/2  PURGE_BACKFILL_DONE %
%   C5:15  PURGE_CYCLE_CTR %
% Rung: 27 %
SOR LIM N9:95 N20:0 N9:91 RES C5:15 EOR
%   N9:95  PURGE_FINAL_VENT %
%   N20:0  PURGE_STATE %
%   N9:91  PURGE_INIT_VENT %
%   C5:15  PURGE_CYCLE_CTR %
% Rung: 28 %
% TITLE: VENT ADSORBERS 2 %
SOR EQU N20:0 N9:97 XIC T4:155/DN LEQ N10:30 N20:5 LEQ N10:33 N20:5 OTE B36:1/4 EOR
%   N20:0  PURGE_STATE %
%   N9:97  PURGE_VENT_ADS_2 %
%   T4:155  STARTUP_DLY %
%   N10:30  ADS_A_INLET_PX_PSIG %
%   N20:5  PURGE_VENT_ADS_2_PX %
%   N10:33  ADS_B_INLET_PX_PSIG %
%   B36:1/4  PURGE_VENT_ADS_2_DN %
% Rung: 29 %
% TITLE: VENT GETTERS 2 %
SOR EQU N20:0 N9:98 XIC T4:155/DN LEQ N10:20 N20:6 OTE B36:1/5 EOR
%   N20:0  PURGE_STATE %
%   N9:98  PURGE_VENT_GET_2 %
%   T4:155  STARTUP_DLY %
%   N10:20  OUTLET_PX_PSIG %
%   N20:6  PURGE_VENT_GET_2_PX %
%   B36:1/5  PURGE_VENT_GET_2_DN %
% Rung: 30 %
% TITLE: FINAL VENT %
SOR EQU N20:0 N9:95 TON T4:107 1.0 30 0 EOR
%   N20:0  PURGE_STATE %
%   N9:95  PURGE_FINAL_VENT %
%   T4:107  PURGE_FINAL_VENT_TM %

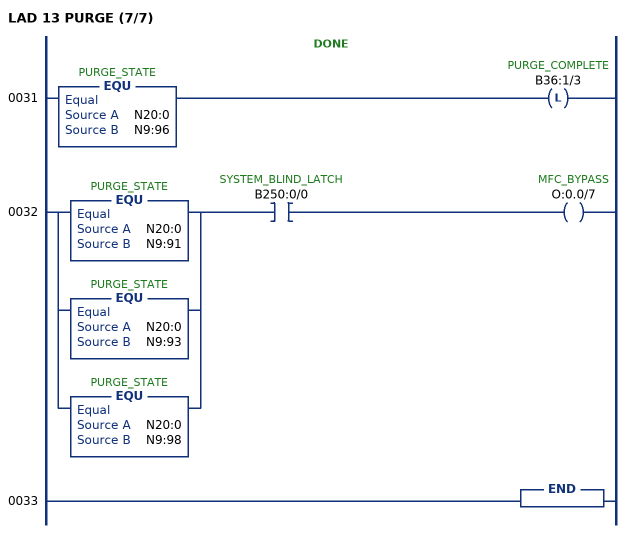
% Rung: 31 %
% TITLE: DONE %
SOR EQU N20:0 N9:96 OTL B36:1/3 EOR
%   N20:0  PURGE_STATE %
%   N9:96  PURGE_DONE %
%   B36:1/3  PURGE_COMPLETE %
% Rung: 32 %
SOR BST EQU N20:0 N9:91 NXB EQU N20:0 N9:93 NXB EQU N20:0 N9:98 BND XIC B250:0/0 OTE O:0.0/7 EOR
%   N20:0  PURGE_STATE %
%   N9:91  PURGE_INIT_VENT %
%   N9:93  PURGE_VENT_GETTER %
%   N9:98  PURGE_VENT_GET_2 %
%   B250:0/0  SYSTEM_BLIND_LATCH %
%   O:0.0/7  MFC_BYPASS %
% Rung: 33 %
SOR END EOR

LADDER 14 "MFM"
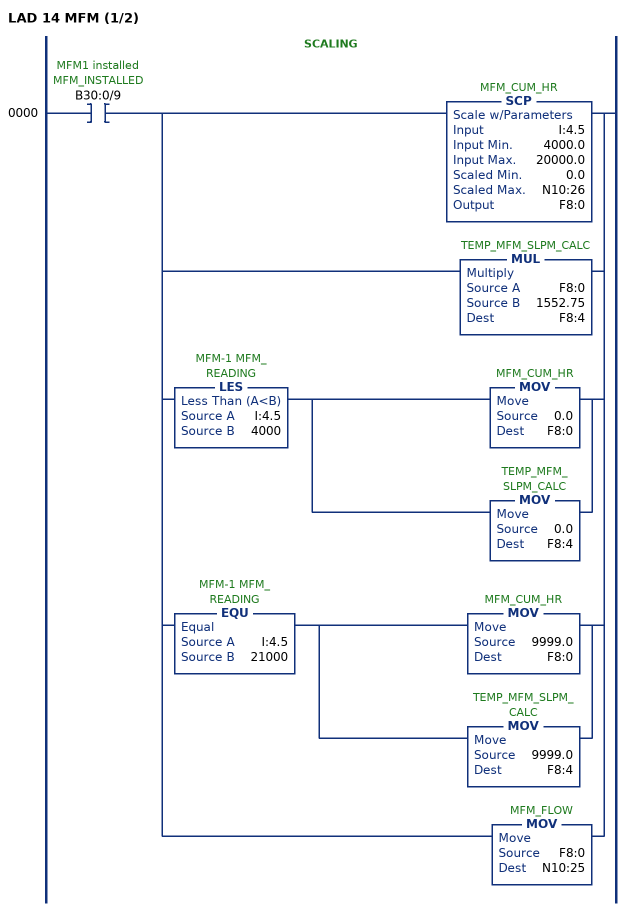
% Rung: 0 %
% TITLE: SCALING %
SOR XIC B30:0/9 BST SCP I:4.5 4000.0 20000.0 0.0 N10:26 F8:0 NXB MUL F8:0 1552.75 F8:4 NXB LES I:4.5 4000 BST MOV 0.0 F8:0 NXB MOV 0.0 F8:4 BND NXB EQU I:4.5 21000 BST MOV 9999.0 F8:0 NXB MOV 9999.0 F8:4 BND NXB MOV F8:0 N10:25 BND EOR
%   B30:0/9  MFM_INSTALLED  "MFM1 installed" %
%   I:4.5  MFM_READING  "MFM-1" %
%   N10:26  MFM_SCALING %
%   F8:0  MFM_CUM_HR %
%   F8:4  TEMP_MFM_SLPM_CALC %
%   N10:25  MFM_FLOW %

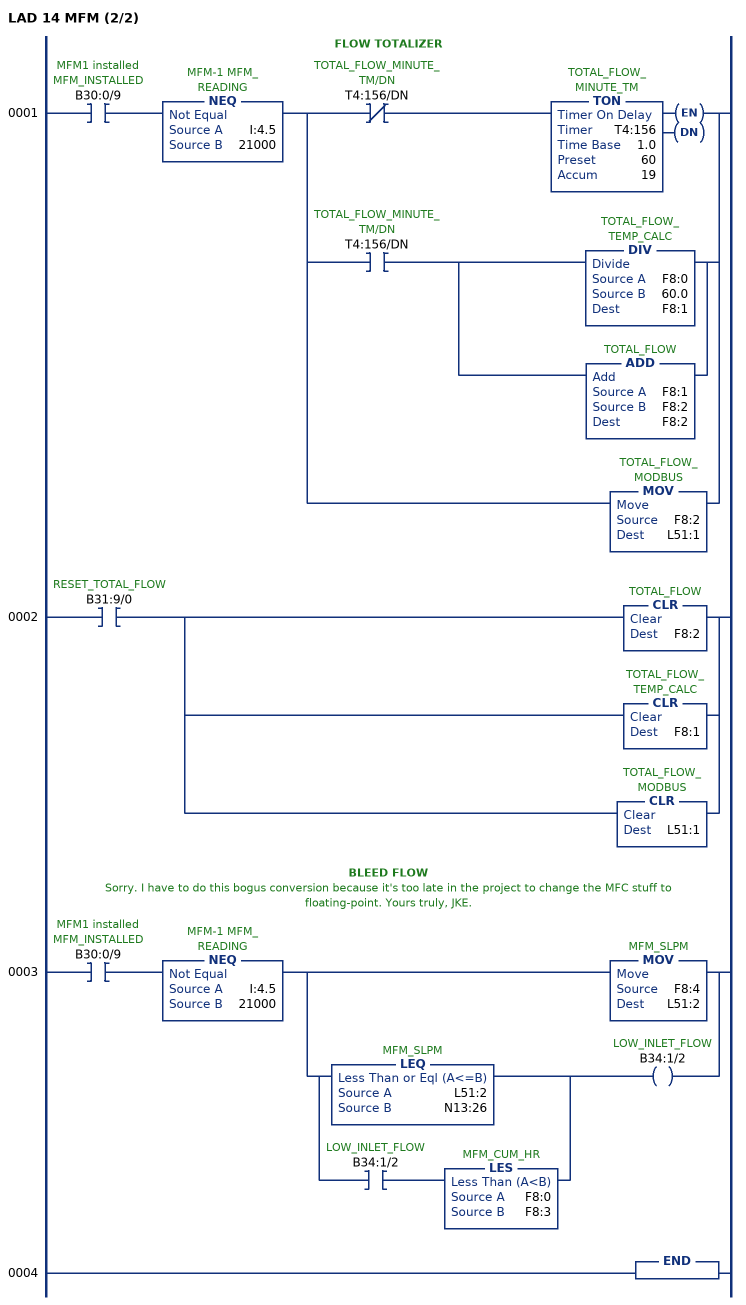
% Rung: 1 %
% TITLE: FLOW TOTALIZER %
SOR XIC B30:0/9 NEQ I:4.5 21000 BST XIO T4:156/DN TON T4:156 1.0 60 19 NXB XIC T4:156/DN BST DIV F8:0 60.0 F8:1 NXB ADD F8:1 F8:2 F8:2 BND NXB MOV F8:2 L51:1 BND EOR
%   B30:0/9  MFM_INSTALLED  "MFM1 installed" %
%   I:4.5  MFM_READING  "MFM-1" %
%   T4:156  TOTAL_FLOW_MINUTE_TM %
%   F8:0  MFM_CUM_HR %
%   F8:1  TOTAL_FLOW_TEMP_CALC %
%   F8:2  TOTAL_FLOW %
%   L51:1  TOTAL_FLOW_MODBUS %
% Rung: 2 %
SOR XIC B31:9/0 BST CLR F8:2 NXB CLR F8:1 NXB CLR L51:1 BND EOR
%   B31:9/0  RESET_TOTAL_FLOW %
%   F8:2  TOTAL_FLOW %
%   F8:1  TOTAL_FLOW_TEMP_CALC %
%   L51:1  TOTAL_FLOW_MODBUS %
% Rung: 3 %
% TITLE: BLEED FLOW %
% Sorry. I have to do this bogus conversion because it's too late in the project to change the MFC stuff to floating-point. Yours truly, JKE. %
SOR XIC B30:0/9 NEQ I:4.5 21000 BST MOV F8:4 L51:2 NXB BST LEQ L51:2 N13:26 NXB XIC B34:1/2 LES F8:0 F8:3 BND OTE B34:1/2 BND EOR
%   B30:0/9  MFM_INSTALLED  "MFM1 installed" %
%   I:4.5  MFM_READING  "MFM-1" %
%   F8:4  TEMP_MFM_SLPM_CALC %
%   L51:2  MFM_SLPM %
%   N13:26  REGEN_BLEED_FLOW %
%   B34:1/2  LOW_INLET_FLOW %
%   F8:0  MFM_CUM_HR %
%   F8:3  BLEED_FLOW_CUTOFF %
% Rung: 4 %
SOR END EOR

LADDER 16 "MFC"
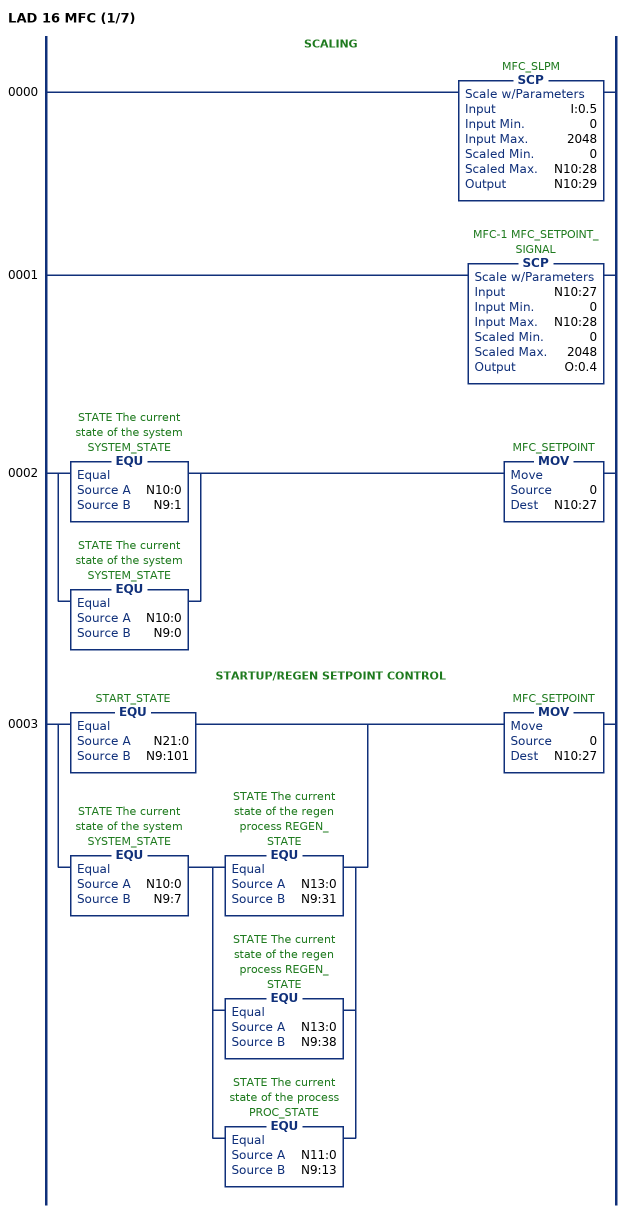
% Rung: 0 %
% TITLE: SCALING %
SOR SCP I:0.5 0 2048 0 N10:28 N10:29 EOR
%   I:0.5  MFC_FEEDBACK  "MFC-1" %
%   N10:28  MFC_SCALING  "in slpm" %
%   N10:29  MFC_SLPM %
% Rung: 1 %
SOR SCP N10:27 0 N10:28 0 2048 O:0.4 EOR
%   N10:27  MFC_SETPOINT %
%   N10:28  MFC_SCALING  "in slpm" %
%   O:0.4  MFC_SETPOINT_SIGNAL  "MFC-1" %
% Rung: 2 %
SOR BST EQU N10:0 N9:1 NXB EQU N10:0 N9:0 BND MOV 0 N10:27 EOR
%   N10:0  SYSTEM_STATE  "STATE The current state of the system" %
%   N9:1  SYSTEM_STANDBY  "STATE System Process" %
%   N9:0  SYSTEM_OFFLINE %
%   N10:27  MFC_SETPOINT %
% Rung: 3 %
% TITLE: STARTUP/REGEN SETPOINT CONTROL %
SOR BST EQU N21:0 N9:101 NXB EQU N10:0 N9:7 BST EQU N13:0 N9:31 NXB EQU N13:0 N9:38 NXB EQU N11:0 N9:13 BND BND MOV 0 N10:27 EOR
%   N21:0  START_STATE %
%   N9:101  START_COOL %
%   N10:0  SYSTEM_STATE  "STATE The current state of the system" %
%   N9:7  SYSTEM_COLD_START %
%   N13:0  REGEN_STATE  "STATE The current state of the regen process" %
%   N9:31  REGEN_DELAY  "STATE Regen Delay" %
%   N9:38  REGEN_DONE %
%   N11:0  PROC_STATE  "STATE The current state of the process" %
%   N9:13  PROC_OVERLAP  "STATE Process Purify Overlap" %
%   N10:27  MFC_SETPOINT %

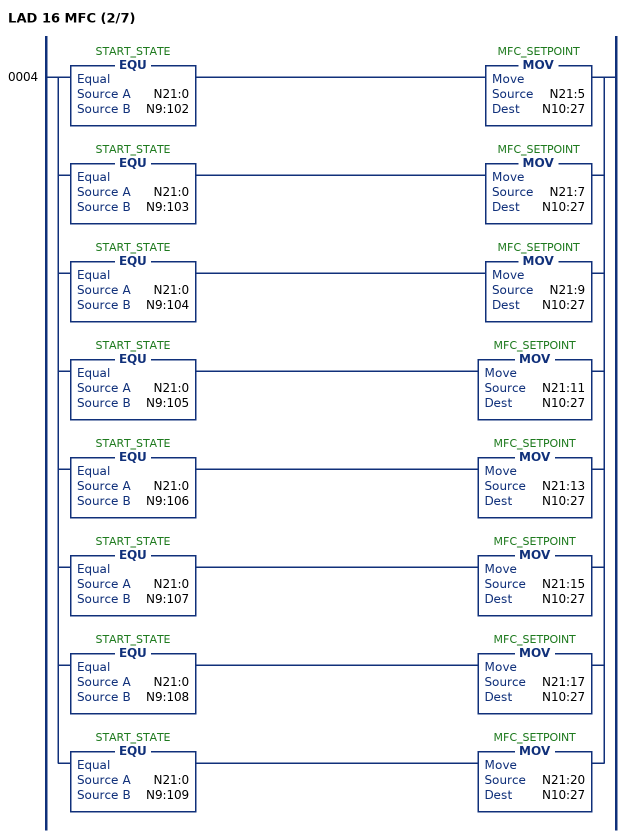
% Rung: 4 %
SOR BST EQU N21:0 N9:102 MOV N21:5 N10:27 NXB EQU N21:0 N9:103 MOV N21:7 N10:27 NXB EQU N21:0 N9:104 MOV N21:9 N10:27 NXB EQU N21:0 N9:105 MOV N21:11 N10:27 NXB EQU N21:0 N9:106 MOV N21:13 N10:27 NXB EQU N21:0 N9:107 MOV N21:15 N10:27 NXB EQU N21:0 N9:108 MOV N21:17 N10:27 NXB EQU N21:0 N9:109 MOV N21:20 N10:27 BND EOR
%   N21:0  START_STATE %
%   N9:102  START_VENT_ADS_1 %
%   N21:5  START_VENT_ADS_1_FLW %
%   N10:27  MFC_SETPOINT %
%   N9:103  START_VENT_GET_1 %
%   N21:7  START_VENT_GET_1_FLW %
%   N9:104  START_HEAT %
%   N21:9  START_HEAT_FLW %
%   N9:105  START_VENT_ALL %
%   N21:11  START_VENT_ALL_FLW %
%   N9:106  START_BACKFILL_1 %
%   N21:13  START_BKFIL_1_FLW %
%   N9:107  START_VENT_ADS_2 %
%   N21:15  START_VENT_ADS_2_FLW %
%   N9:108  START_VENT_GET_2 %
%   N21:17  START_VENT_GET_2_FLW %
%   N9:109  START_BACKFILL_2 %
%   N21:20  START_BKFIL_2_FLW %

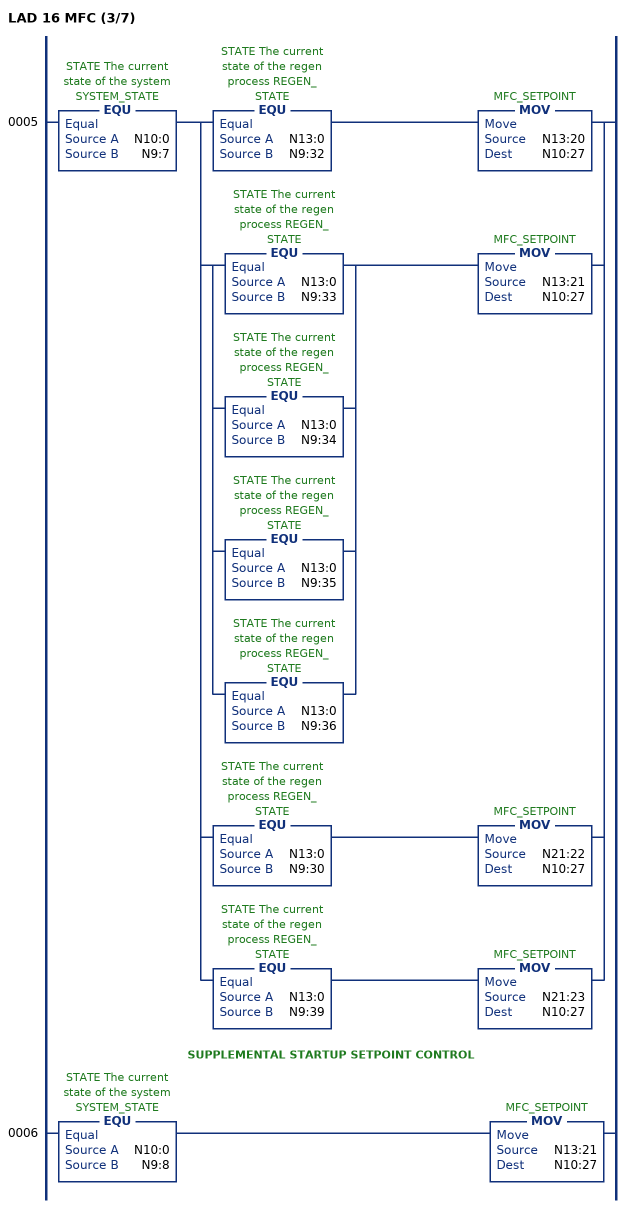
% Rung: 5 %
SOR EQU N10:0 N9:7 BST EQU N13:0 N9:32 MOV N13:20 N10:27 NXB BST EQU N13:0 N9:33 NXB EQU N13:0 N9:34 NXB EQU N13:0 N9:35 NXB EQU N13:0 N9:36 BND MOV N13:21 N10:27 NXB EQU N13:0 N9:30 MOV N21:22 N10:27 NXB EQU N13:0 N9:39 MOV N21:23 N10:27 BND EOR
%   N10:0  SYSTEM_STATE  "STATE The current state of the system" %
%   N9:7  SYSTEM_COLD_START %
%   N13:0  REGEN_STATE  "STATE The current state of the regen process" %
%   N9:32  REGEN_VENT  "STATE Regen Vent" %
%   N13:20  REGEN_VENT_FLOW %
%   N10:27  MFC_SETPOINT %
%   N9:33  REGEN_HEAT_BED  "STATE Regen Heat wall" %
%   N9:34  REGEN_RUN  "STATE Regen Running" %
%   N9:35  REGEN_COOL_WALL  "STATE Regen Cool wall" %
%   N9:36  REGEN_COOL  "STATE Regen Cool" %
%   N13:21  REGEN_MAIN_FLOW %
%   N9:30  REGEN_STANDBY  "STATE Regen Standby" %
%   N21:22  START_REG_BLEED_FLW %
%   N9:39  REGEN_BACKFILL %
%   N21:23  START_REG_BKFIL_FLW %
% Rung: 6 %
% TITLE: SUPPLEMENTAL STARTUP SETPOINT CONTROL %
SOR EQU N10:0 N9:8 MOV N13:21 N10:27 EOR
%   N10:0  SYSTEM_STATE  "STATE The current state of the system" %
%   N9:8  SYSTEM_SUPPLEMENTAL %
%   N13:21  REGEN_MAIN_FLOW %
%   N10:27  MFC_SETPOINT %

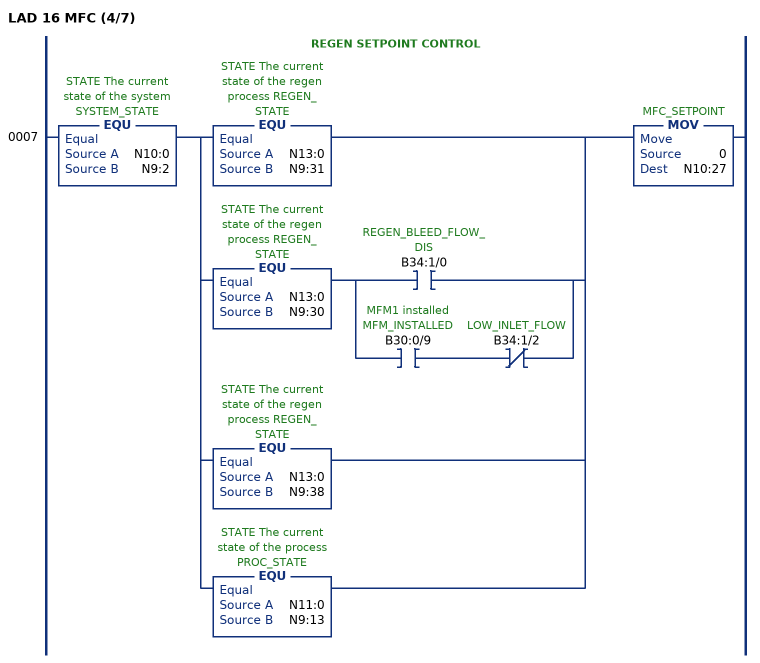
% Rung: 7 %
% TITLE: REGEN SETPOINT CONTROL %
SOR EQU N10:0 N9:2 BST EQU N13:0 N9:31 NXB EQU N13:0 N9:30 BST XIC B34:1/0 NXB XIC B30:0/9 XIO B34:1/2 BND NXB EQU N13:0 N9:38 NXB EQU N11:0 N9:13 BND MOV 0 N10:27 EOR
%   N10:0  SYSTEM_STATE  "STATE The current state of the system" %
%   N9:2  SYSTEM_PROCESS  "STATE System Process" %
%   N13:0  REGEN_STATE  "STATE The current state of the regen process" %
%   N9:31  REGEN_DELAY  "STATE Regen Delay" %
%   N9:30  REGEN_STANDBY  "STATE Regen Standby" %
%   B34:1/0  REGEN_BLEED_FLOW_DIS %
%   B30:0/9  MFM_INSTALLED  "MFM1 installed" %
%   B34:1/2  LOW_INLET_FLOW %
%   N9:38  REGEN_DONE %
%   N11:0  PROC_STATE  "STATE The current state of the process" %
%   N9:13  PROC_OVERLAP  "STATE Process Purify Overlap" %
%   N10:27  MFC_SETPOINT %

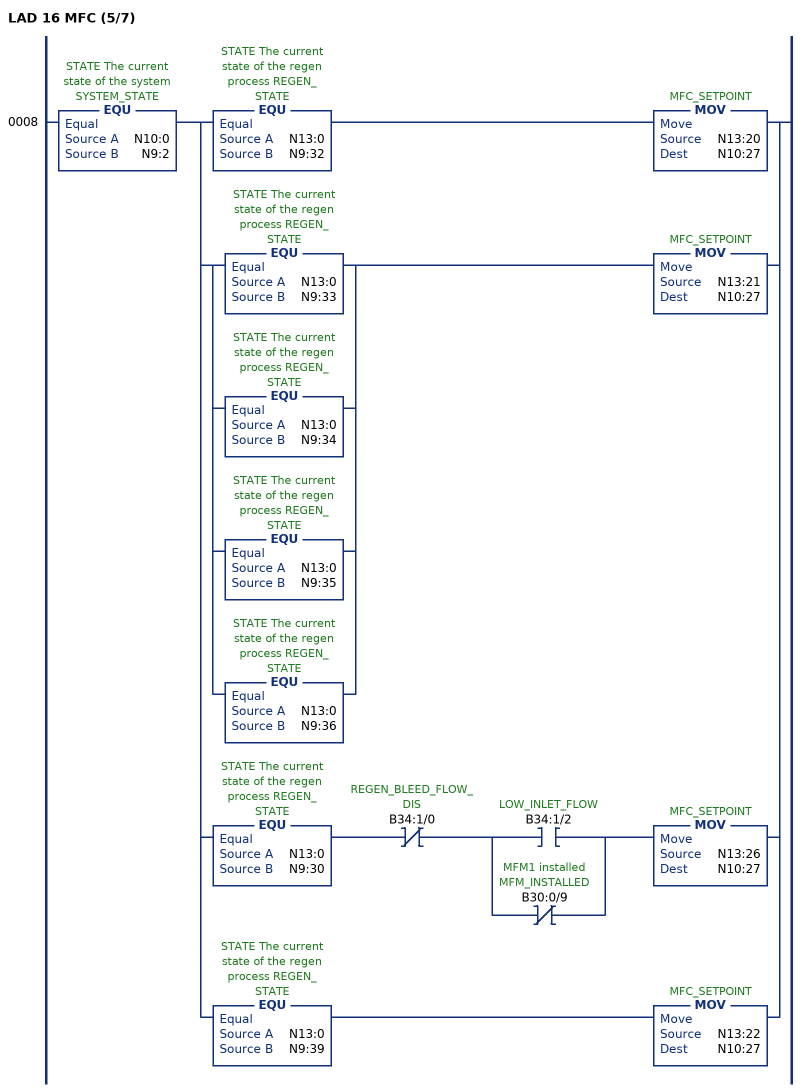
% Rung: 8 %
SOR EQU N10:0 N9:2 BST EQU N13:0 N9:32 MOV N13:20 N10:27 NXB BST EQU N13:0 N9:33 NXB EQU N13:0 N9:34 NXB EQU N13:0 N9:35 NXB EQU N13:0 N9:36 BND MOV N13:21 N10:27 NXB EQU N13:0 N9:30 XIO B34:1/0 BST XIC B34:1/2 NXB XIO B30:0/9 BND MOV N13:26 N10:27 NXB EQU N13:0 N9:39 MOV N13:22 N10:27 BND EOR
%   N10:0  SYSTEM_STATE  "STATE The current state of the system" %
%   N9:2  SYSTEM_PROCESS  "STATE System Process" %
%   N13:0  REGEN_STATE  "STATE The current state of the regen process" %
%   N9:32  REGEN_VENT  "STATE Regen Vent" %
%   N13:20  REGEN_VENT_FLOW %
%   N10:27  MFC_SETPOINT %
%   N9:33  REGEN_HEAT_BED  "STATE Regen Heat wall" %
%   N9:34  REGEN_RUN  "STATE Regen Running" %
%   N9:35  REGEN_COOL_WALL  "STATE Regen Cool wall" %
%   N9:36  REGEN_COOL  "STATE Regen Cool" %
%   N13:21  REGEN_MAIN_FLOW %
%   N9:30  REGEN_STANDBY  "STATE Regen Standby" %
%   B34:1/0  REGEN_BLEED_FLOW_DIS %
%   B34:1/2  LOW_INLET_FLOW %
%   B30:0/9  MFM_INSTALLED  "MFM1 installed" %
%   N13:26  REGEN_BLEED_FLOW %
%   N9:39  REGEN_BACKFILL %
%   N13:22  REGEN_BACKFILL_FLOW %

